{attribute 'qualified_only'}
{attribute 'strict'}
{attribute 'to_string'}
TYPE ProcessExecution_e :
(
	ExecuteImmediately,
	ExecuteWithPrevious,
	_MAX
);
END_TYPE

(* stored: Version 1.1.0.1, ProductVersion 3.1.4024.6
   EnumerationTextList ProcessExecution_e: Id {ca5b2402-e281-4d2a-a2c7-282e5c601458} *)
